FUNCTION_BLOCK IntQueue
VAR
	elements : FB_BA_DynamicArray := (uiEntrySize := SIZEOF(INT), uiMinExpCount := 4);
	length : USINT := 0;
END_VAR

METHOD clear : BOOL
VAR_INPUT
END_VAR
elements.Reset();
length := 0;
END_METHOD

METHOD contains : BOOL
VAR_INPUT
	value : INT;
END_VAR
VAR_INST
	i : INT;
END_VAR
IF length = 0 THEN
	contains := FALSE;
	RETURN;
END_IF

FOR i:=0 TO length-1 BY 1 DO
	IF get(i) = value THEN
		contains := TRUE;
		RETURN;
	END_IF
END_FOR
contains := FALSE;
END_METHOD

METHOD get : INT
VAR_INPUT
	i : INT;
END_VAR
elements.GetEntry(diIndex := i, pResultEntry := ADR(get));
END_METHOD

METHOD isEmpty : BOOL
VAR_INPUT
END_VAR
isEmpty := (length = 0);
END_METHOD

METHOD poll : INT
VAR_INST
	temp : INT;
	i : INT;
END_VAR
temp := get(i := 0);
elements.RemoveEntry(diIndex := 0);
length := length - 1;
poll := temp;
END_METHOD

METHOD push : BOOL
VAR_INPUT
	value : INT;
END_VAR
elements.AddEntry(pEntry := ADR(value));
length := length + 1;
END_METHOD

METHOD set : BOOL
VAR_INPUT
	i : INT;
	value : INT;
END_VAR
elements.SetEntry(i, ADR(value));
END_METHOD

METHOD size : USINT
VAR_INPUT
END_VAR
size := length;
END_METHOD

METHOD sort : BOOL
VAR_INPUT
END_VAR
VAR_INST
	i : INT;
	j : INT;
	temp : INT;
END_VAR
FOR i:=0 TO GVL.maxMaterials BY 1 DO
	FOR j:=0 TO GVL.maxMaterials BY 1 DO
		IF get(j) > get(j+1) THEN //swap
			temp := get(j);
			set(j, get(j+1));
			set(j+1, temp);
		END_IF
	END_FOR
END_FOR
END_METHOD

END_FUNCTION_BLOCK

(* stored: Version 1.1.0.1, ProductVersion 3.1.4024.11
   POU IntQueue: Id {b88eabe4-fa96-488a-9c59-79d0926b2421}, SpecialFunc None
   Method clear: Id {e2568c0d-1a27-4165-868b-001d96ffa635}
   Method contains: Id {1ea2cef5-ff89-4cb3-8414-f91e89824126}
   Method get: Id {f77f5f86-6803-4a8e-a82e-15512b7a2d13}
   Method isEmpty: Id {2e909f5b-f462-464b-a4f4-530341b5a502}
   Method poll: Id {d7ffe0bd-a70d-474f-b52b-bb90a8761c71}
   Method push: Id {4f38a899-fe5c-4539-b0ae-ab2eb4fd4d3f}
   Method set: Id {6e48312b-26e4-4a4f-893e-4e19c9cf9369}
   Method size: Id {af0b9551-be39-498e-a520-c313ac29b4d9}
   Method sort: Id {b819151d-789f-45e6-abe7-8db18aa34d47} *)
